FUNCTION_BLOCK FB_Rain_Generator
VAR_INPUT
	_gen : BOOL;
	_time : TOD;
END_VAR
VAR_OUTPUT
	_rain : BOOL;
END_VAR
VAR
END_VAR

END_FUNCTION_BLOCK

(* stored: Version 1.1.0.1, ProductVersion 3.1.4018.5
   POU FB_Rain_Generator: Id {1ccdcf26-6c06-41e3-9459-9b74abed1569}, SpecialFunc None *)
